# B&R Automation Studio project Haus
Automation Studio 4.8.4.50 SP; technology packages: mapp 5.13.1, mappView 5.13.1

## Configuration iCMSLight

CPU X20CP1586, AutomationRuntime B4.82, Build 4.1.2, Safety 0.0

### Task classes (Cpu.sw)
```
Cyclic#4 (cycle 32000 us, tolerance 32000 us):
  Solarpumpe <- Haus.Solarpumpe.prg
  Garage <- Haus.Garage.prg
  ErrorHandl <- Haus.ErrorHandling.prg
Cyclic#6 (cycle 256000 us, tolerance 256000 us):
  Main <- Haus.Main.prg
  Datenverwa <- Haus.Datenverwaltung.prg
DataObjects: assl3, Acp10sys, assl2, assl1
Binaries: TCLang, udbdef, mvLoader, TCData, arsvcreg, User, arconfig, Role, iomap, asfw, ashwac, ashwd, sysconf, Speicher, Units, RollenDB, Alarme, Config, VehicleAla, History, asnxdb2, OpcUaMap, MR4, Acp10map, acp10cfg, Shuttle2, MainAlarme, Alarm
Libraries: standard, runtime, operator, sys_lib, astime, brsystem, Convert, AsBrStr, ksTime, MpBase, FileIO, MpServer, AsMath, MpCom, MpRecipe, ksStpHist, DataObj, aruser, arssl, AsTCP, ksBuffer, AsOpcUac, AsHttp, MTBasics, AsHydCon, dvframe, MTTypes, AsUDP, ArCan, MTProfile, powerlnk, ksAlarm, MpAlarmX, AsSMTP, asstring
```

### Hardware
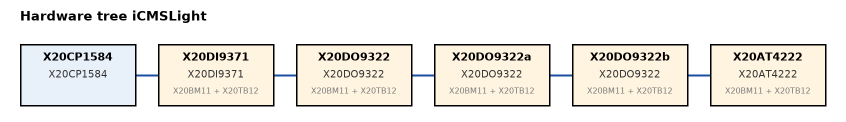
```
X20AT4222 : X20AT4222 v1.3.0.0  [SS1 -> X20TB12b.SS; SL -> X20BM11b.SL1]
  Supervision = off
  SensorType04 = off
X20BM11 : X20BM11 v1.0.0.1  [X2X1 -> X20BM11a.X2X2]
X20BM11a : X20BM11 v1.0.0.1  [X2X1 -> X20CP1584.IF6]
X20BM11b : X20BM11 v1.0.0.1  [X2X1 -> X20BM11d.X2X2]
X20BM11c : X20BM11 v1.0.0.1  [X2X1 -> X20BM11.X2X2]
X20BM11d : X20BM11 v1.0.0.1  [X2X1 -> X20BM11c.X2X2]
X20CP1584 : X20CP1584 v1.8.0.0
  Connector IF2:
    ActivateDevice = 1
    Mode = Manual
    InternetAddress = 192.168.0.101
    SubnetMask = 255.255.0.0
    ActivateOSAFT = 1
    OSAFTPortNumber = 10003
  Connector IF3:
    ActivatePowerlink = 0
  ConfigurationID = Haus
  SimulationModeOpcUa = off
  RemanentGlobalPvSize = 120652
  VolatileGlobalPvSize = 300000
  Connections = 10
  IdleTaskClass = 6
  TaskClassIdleTime = 10000
  CyclicTaskClassCount = 6
  Cyclic1Duration = 2000
  Cyclic1Tolerance = 2000
  Cyclic2Duration = 8000
  Cyclic2Tolerance = 8000
  Cyclic3Duration = 16000
  Cyclic3Tolerance = 16000
  Cyclic4Duration = 32000
  Cyclic4Tolerance = 32000
  Cyclic5Duration = 128000
  Cyclic5Tolerance = 128000
  Cyclic6Duration = 256000
  Cyclic6Tolerance = 256000
  FileDevice1
  FileDeviceName1 = Home
  FileDevicePath1 = C:\
  FileDevice2
  FileDeviceName2 = Alarm
  FileDevicePath2 = C:\Alarm
  FileDevice3
  FileDeviceName3 = Datenverwaltung
  FileDevicePath3 = C:\Datenverwaltung
  FileDevice4
  FileDeviceName4 = Logger
  FileDevicePath4 = C:\Logger
  TimeZone = 140
  ActivateDaylightSavingTime = 1
  FtpUser1
  FtpUsername1 = kssr
  FtpUserPassword1 = Z4sCxg1Qn6GbuX9/lK+IGbQPtWBLs+BxMSzu+/HSn5M=
  FtpUserSalt1 = QM4eEhG1
  FTPAccessRight1 = 0
  FTPdevice1 = ALL
  ActivateOpcUa = 1
  OpcUaLimitsMaxSessions = 0
  OpcUaLimitsMaxBrowseContinuationPoints = 50
  OpcUaInformationModels_PV_Version = 2
X20DI9371 : X20DI9371 v1.1.0.0  [SS1 -> X20TB12a.SS; SL -> X20BM11a.SL1]
  Supervision = off
X20DO9322 : X20DO9322 v1.2.0.0  [SS1 -> X20TB12.SS; SL -> X20BM11.SL1]
  Supervision = off
X20DO9322a : X20DO9322 v1.2.0.0  [SS1 -> X20TB12c.SS; SL -> X20BM11c.SL1]
  Supervision = off
X20DO9322b : X20DO9322 v1.2.0.0  [SS1 -> X20TB12d.SS; SL -> X20BM11d.SL1]
  Supervision = off
X20TB12 : X20TB12 v1.0.0.0
X20TB12a : X20TB12 v1.0.0.0
X20TB12b : X20TB12 v1.0.0.0
X20TB12c : X20TB12 v1.0.0.0
X20TB12d : X20TB12 v1.0.0.0
```

### IoMap.iom - X20CP1584/IoMap.iom
```iecst
VAR_CONFIG
	::Garage:IO.Output.Command AT %QX."X20DO9322".DigitalOutput01;
	::Garage:IO.Input.Opened AT %IX."X20DI9371".DigitalInput01;
	::Garage:IO.Input.Closed AT %IX."X20DI9371".DigitalInput02;
	::Solarpumpe:IO.Input.DachTemp AT %IW."X20AT4222".Temperature01;
	::Solarpumpe:IO.Input.RuecklaufTemp AT %IW."X20AT4222".Temperature02;
	::Solarpumpe:IO.Input.KesselTemp AT %IW."X20AT4222".Temperature03;
	::Garage:IO.Input.Button AT %IX."X20DI9371".DigitalInput03;
	::Solarpumpe:IO.Output.PumpeUp  AT %QX."X20DO9322a".DigitalOutput01;
	::Solarpumpe:IO.Output.PumpeDown  AT %QX."X20DO9322a".DigitalOutput02;
END_VAR
```

### Alarm.mpalarmxcore - X20CP1584/mappServices/Alarm.mpalarmxcore
```
Element gAlarmXCore (Type=mpalarmxcore)
  mapp.AlarmX.Core:
    Mapping:
      [0]
  mapp.AlarmX.Core.Configuration:
    [0]:
      Name = GarageUndefined
      Message = Das Garagentor ist in einem undefiniertem Zustand
      Behavior = PersistentAlarm
    [1]:
      Name = PumpUpNotActive
      Message = Die &#x2B06; Pumpe wurde nicht aktiviert da die Rücklauftemperatur zu hoch ist.
      Severity = 2
      Behavior = PersistentAlarm
  mapp.AlarmX.Core.Queries:
    [0]:
      Name = ActiveErrors
      Update = ::ErrorHandl:ActiveAlarms.Error.UpdateFlag
      Source:
        SELECT:
          [0]:
            Column = Severity
            PV = ::ErrorHandl:ActiveAlarms.Error.ActiveAlarms[]
        WHERE:
          [0]:
            Column = Severity
            CompareTo:
              Value = 1
    [1]:
      Name = ActiveWarnings
      Update = ::ErrorHandl:ActiveAlarms.Warning.UpdateFlag
      Source:
        SELECT:
          [0]:
            Column = Severity
            PV = ::ErrorHandl:ActiveAlarms.Warning.ActiveAlarms[]
        WHERE:
          [0]:
            Column = Severity
            CompareTo:
              Value = 2
    [2]:
      Name = ActiveInfos
      Update = ::ErrorHandl:ActiveAlarms.Info.UpdateFlag
      Source:
        SELECT:
          [0]:
            Column = Severity
            PV = ::ErrorHandl:ActiveAlarms.Info.ActiveAlarms[]
        WHERE:
          [0]:
            Column = Severity
            CompareTo:
              Value = 3
  mapp.AlarmX.Core.Categories:
    [0]:
      Name = Error
      SourceProperty:
        Severity = 1
    [1]:
      Name = Warning
      SourceProperty:
        Severity = 2
    [2]:
      Name = Info
      SourceProperty:
        Severity = 3
```

## Logical view

Binary libraries used (declarations not repeated): operator, runtime, astime, sys_lib, brsystem, standard, Convert, AsBrStr, ksTime 1.04.0, FileIO, AsMath, MpServer 5.13.0, MpBase 5.13.0, MpRecipe 5.13.1, MpCom 5.13.1, DataObj, MpAlarmX 5.11.2, AsSMTP, asstring

### Global.var - Global variables
```iecst
VAR
	gCurrentDT : DATE_AND_TIME := DT#1970-01-01-00:00:00;
	gSmtpSend : SmtpSend := (0);
	gCurrentDTStruct : DTStructure := (0);
END_VAR
```

### Package Logical/Libraries - Global libraries

### Library Logical/Libraries/ksStpHist (ANSIC, version 1.00.0) - Step History Baustein
Depends on: standard

#### ksStpHist.typ
```iecst
TYPE
	KsStepData_type : 	STRUCT
		Last : DINT;
		Act : DINT;
		Next : DINT; (*nur für single step*)
		Reset : DINT; (*step after reset*)
	END_STRUCT;
	ksStepHistoryEntry : 	STRUCT
		Act : USINT;
		ET : TIME;
	END_STRUCT;
END_TYPE
```

#### ksStpHist.fun
```iecst
{REDUND_ERROR} FUNCTION_BLOCK ksStepHistory (*speichert Schritthistorie*) (*$GROUP=User,$CAT=User,$GROUPICON=User.png,$CATICON=User.png*)
	VAR_INPUT
		in_Step : {REDUND_UNREPLICABLE} KsStepData_type;
		in_ET : {REDUND_UNREPLICABLE} TIME;
	END_VAR
	VAR
		aData : {REDUND_UNREPLICABLE} ARRAY[0..MAX_IDX_STEP_HISTORY_ENTRIES] OF ksStepHistoryEntry;
		i : {REDUND_UNREPLICABLE} USINT;
		Last : USINT;
	END_VAR
END_FUNCTION_BLOCK
```

#### ksStpHist.var
```iecst
VAR CONSTANT
	MAX_IDX_STEP_HISTORY_ENTRIES : USINT := 95;
END_VAR
```

#### ksStpHist.c
```c
#include <bur/plctypes.h>
#ifdef __cplusplus
	extern "C"
	{
#endif
	#include "ksStpHist.h"
#ifdef __cplusplus
	};
#endif
/* speichert Schritthistorie */
void ksStepHistory(struct ksStepHistory* inst)
{
	if (inst->i >= MAX_IDX_STEP_HISTORY_ENTRIES)
	{
		inst->i = 0;
	}

	if (inst->in_Step.Act != inst->in_Step.Next)
	{
		inst->aData[inst->i].Act = inst->in_Step.Act;
		inst->aData[inst->i].ET = inst->in_ET;
		inst->i++;
	}

}
```

### Program Logical/Haus/Main (ANSIC)

#### Main.c - Init, cyclic, exit code
```c
#include <bur/plctypes.h>
#include <stdbool.h>

#ifdef _DEFAULT_INCLUDES
	#include <AsDefault.h>
#endif

void _INIT ProgramInit(void)
{

}

void _CYCLIC ProgramCyclic(void)
{
	DTGetTime_1.enable = true;
	DTGetTime(&DTGetTime_1);

	gCurrentDT = DTGetTime_1.DT1;

	DT_TO_DTStructure(gCurrentDT, (UDINT)&gCurrentDTStruct);

	//Email Sender initialisieren

//	gSmtpSend.enable= true;
	gSmtpSend.pHost= (UDINT)"smtp.gmail.com";
	gSmtpSend.pSender= (UDINT)"sdillinger.tai@gmail.com";
	gSmtpSend.pReceiver= (UDINT)"mihawk14@web.de";
	gSmtpSend.pSubject= (UDINT)"test";
	gSmtpSend.pText= (UDINT)"test";
//	gSmtpSend.pUser = (UDINT)"sdillinger.tai@gmail.com";
//	gSmtpSend.pPassword= ADR(gMAIL.smpt_pw) // 'mein GMX Passwort'
//	gSmtpSend.pAttachment= ADR(AttStruc) // momentan 0
//	gSmtpSend.pDomain= 0
//	gSmtpSend.pSecurity= 0
//	gSmtpSend.timeout= 0
	gSmtpSend.port = 465; // 485,0, 0der 25
//	SmtpSend(&gSmtpSend);
}

void _EXIT ProgramExit(void)
{

}
```

#### Main.var - Local variables
```iecst
VAR
	DTGetTime_1 : DTGetTime := (0);
END_VAR
```

### Program Logical/Haus/Datenverwaltung (ANSIC)

#### Datenverwaltung.c - Init, cyclic, exit code
```c
#include <bur/plctypes.h>
#include <stdbool.h>
#include <AsBrStr.h>

#ifdef _DEFAULT_INCLUDES
	#include <AsDefault.h>
#endif

void _INIT ProgramInit(void)
{
    DirCreate_DV.enable = true;
    DirCreate_DV.pDevice = (UDINT)"Home";
    DirCreate_DV.pName = (UDINT)"Datenverwaltung";
    DirCreate(&DirCreate_DV);

    DTGetTime_DV.enable = true;
    DTGetTime(&DTGetTime_DV);

    Visu.StatusTime = DTGetTime_DV.DT1;
    brsstrcpy((UDINT)Visu.StatusText, (UDINT)"Steuerung neu gestartet");

    FileInfo_0.enable = true;
    FileInfo_0.pDevice = (UDINT)"Datenverwaltung";
    FileInfo_0.pName = (UDINT)"DV.csv";
    FileInfo_0.pInfo = (UDINT)&pFileInfo;
    FileInfo(&FileInfo_0);

    Visu.Load = true;

}

void _CYCLIC ProgramCyclic(void)
{
    DTGetTime_DV.enable = true;
    DTGetTime(&DTGetTime_DV);

    MpRecipeCsv_DV.MpLink = &gRecipeCsv;
    MpRecipeCsv_DV.Enable = true;
    MpRecipeCsv_DV.Save = Visu.Save;
    MpRecipeCsv_DV.Load = Visu.Load;
    MpRecipeCsv_DV.DeviceName = (UDINT)"Datenverwaltung";
    MpRecipeCsv_DV.FileName = (UDINT)"DV";
    MpRecipeCsv(&MpRecipeCsv_DV);

    for(i=0;i<=MAX_DV;i++)
    {
        MpRecipeRegPar_DV[i].MpLink = &gRecipeCsv;
        MpRecipeRegPar_DV[i].Enable = true;
        MpRecipeRegPar_DV[i].PVName = (UDINT)&PVNames[i];
        MpRecipeRegPar(&MpRecipeRegPar_DV[i]);
    }

    switch(State)
    {
        case STATE_DV_WAIT:
            Visu.ButtonAktiv = true;
            if(Visu.Save)
            {
                Visu.ButtonAktiv = false;
                State = STATE_DV_SAVE;
            }
            else if(Visu.Load)
            {
                Visu.ButtonAktiv = false;
                State = STATE_DV_LOAD;
            }

            break;

        case STATE_DV_SAVE:
            if(MpRecipeCsv_DV.CommandDone)
            {
                Visu.StatusTime = DTGetTime_DV.DT1;
                brsstrcpy((UDINT)Visu.StatusText, (UDINT)"Speichern abgeschlossen");
                Visu.Save = false;
                State = STATE_DV_WAIT;
            }

            break;

        case STATE_DV_LOAD:
            if(MpRecipeCsv_DV.CommandDone)
            {
                Visu.StatusTime = DTGetTime_DV.DT1;
                brsstrcpy((UDINT)Visu.StatusText, (UDINT)"Laden abgeschlossen");
                Visu.Load = false;
                State = STATE_DV_WAIT;
            }

            break;

    }

}

void _EXIT ProgramExit(void)
{
    MpRecipeCsv_DV.Enable = false;
    MpRecipeCsv(&MpRecipeCsv_DV);

//    for(i=0;i<=MAX_DV;i++)
//    {
//        MpRecipeRegPar_DV[i].Enable = false;
//        MpRecipeRegPar(&MpRecipeRegPar_DV[i]);
//    }
}
```

#### Datenverwaltung.typ - Local data types
```iecst
TYPE
	STATE_DV_enum :
		(
		STATE_DV_WAIT,
		STATE_DV_SAVE,
		STATE_DV_LOAD
		);
	DatenverwaltungVisu_typ : 	STRUCT
		Save : BOOL;
		Load : BOOL;
		ButtonAktiv : BOOL;
		StatusText : STRING[255];
		StatusTime : DATE_AND_TIME;
	END_STRUCT;
END_TYPE
```

#### Datenverwaltung.var - Local variables
```iecst
VAR CONSTANT
	MAX_DV : USINT := 10;
END_VAR
VAR
	MpRecipeRegPar_DV : ARRAY[0..MAX_DV] OF MpRecipeRegPar := [11((0))];
	MpRecipeCsv_DV : MpRecipeCsv := (0);
	PVNames : ARRAY[0..MAX_DV] OF STRING[255] := ['Solarpumpe:DachSollTemp','Solarpumpe:KesselSollTemp','Solarpumpe:RuecklaufSollTemp','RuecklaufTimeOffset',7('')];
	DTGetTime_DV : DTGetTime := (0);
	DirCreate_DV : DirCreate := (0);
	i : USINT := 0;
	Visu : DatenverwaltungVisu_typ := (0);
	State : STATE_DV_enum := STATE_DV_WAIT;
	FileInfo_0 : FileInfo := (0);
	pFileInfo : REFERENCE TO fiFILE_INFO;
END_VAR
```

### Program Logical/Haus/Solarpumpe (ANSIC)

#### Solarpumpe.c - Init, cyclic, exit code
```c
#include <bur/plctypes.h>
#include <stdbool.h>

#ifdef _DEFAULT_INCLUDES
	#include <AsDefault.h>
#endif

void _INIT ProgramInit(void)
{

}

void _CYCLIC ProgramCyclic(void)
{
	if(IO.Output.PumpeDown)
		brsstrcpy((UDINT)Visu.PumpeDownStyle, (UDINT)"StatusOk");
	else
		brsstrcpy((UDINT)Visu.PumpeDownStyle, (UDINT)"StatusNOk");

	if(IO.Output.PumpeUp)
		brsstrcpy((UDINT)Visu.PumpeUpStyle, (UDINT)"StatusOk");
	else
		brsstrcpy((UDINT)Visu.PumpeUpStyle, (UDINT)"StatusNOk");

	UDINTTimeOffset = Mem.RuecklaufTimeOffset;

	TON_PumpUp.IN = IO.Output.PumpeDown;
	TON_PumpUp.PT = UDINTTimeOffset * 1000;
	TON(&TON_PumpUp);

	R_TRIG_Start.CLK = IO.Output.PumpeUp && IO.Output.PumpeDown;
	R_TRIG(&R_TRIG_Start);

	R_TRIG_Stop.CLK = !(IO.Output.PumpeUp && IO.Output.PumpeDown);
	R_TRIG(&R_TRIG_Stop);

	if(R_TRIG_Start.Q)
	{
		Info.LastStart = gCurrentDT;
	}

	if(R_TRIG_Stop.Q)
	{
	 	Info.LastStop = gCurrentDT;
		Info.LaufzeitDownAkt = 0;
		Info.LaufzeitUpAkt = 0;
	}

	if(Mem.Aktiv)
	{
		if(IO.Input.DachTemp >= Mem.DachSollTemp && IO.Input.KesselTemp <= Mem.KesselSollTemp)
		{
			IO.Output.PumpeDown = true;
			Info.LaufzeitDownAkt += CURRENT_CYCLE_TIME;
			Info.LaufzeitUpGes += CURRENT_CYCLE_TIME;

			if(TON_PumpUp.Q)
			{
				if(IO.Input.RuecklaufTemp <= Mem.RuecklaufSollTemp)
				{
					IO.Output.PumpeUp = true;
					Info.LaufzeitUpAkt += CURRENT_CYCLE_TIME;
					Info.LaufzeitDownGes += CURRENT_CYCLE_TIME;

					MpAlarmXReset(&gAlarmXCore, "PumpUpNotActive");
				}
				else
				{
					MpAlarmXSet(&gAlarmXCore, "PumpUpNotActive");
				}
			}
		}
		else
		{
			IO.Output.PumpeDown = false;
			IO.Output.PumpeUp = false;
		}

	}
	else
	{
		IO.Output.PumpeDown = false;
		IO.Output.PumpeUp = false;
	}
}

void _EXIT ProgramExit(void)
{

}
```

#### Solarpumpe.typ - Local data types
```iecst
TYPE
	SolarpumpeIO_typ : 	STRUCT
		Input : SolarpumpeInputs_typ;
		Output : SolarpumpeOutputs_typ;
	END_STRUCT;
	SolarpumpeInputs_typ : 	STRUCT
		DachTemp : INT;
		RuecklaufTemp : INT;
		KesselTemp : INT;
	END_STRUCT;
	SolarpumpeOutputs_typ : 	STRUCT
		PumpeDown : BOOL;
		PumpeUp : BOOL;
	END_STRUCT;
	SolarpumpeVisu_typ : 	STRUCT
		PumpeUpStyle : STRING[99];
		PumpeDownStyle : STRING[99];
	END_STRUCT;
	SolarpumpeInfo_typ : 	STRUCT
		LaufzeitDownAkt : DINT;
		LaufzeitUpAkt : DINT;
		LaufzeitDownGes : DINT;
		LaufzeitUpGes : DINT;
		LastStart : DATE_AND_TIME;
		LastStop : DATE_AND_TIME;
	END_STRUCT;
	SolarpumpeMem_typ : 	STRUCT
		DachSollTemp : INT;
		KesselSollTemp : INT;
		RuecklaufSollTemp : INT;
		Aktiv : BOOL;
		RuecklaufTimeOffset : DATE_AND_TIME;
	END_STRUCT;
END_TYPE
```

#### Solarpumpe.var - Local variables
```iecst
VAR
	IO : SolarpumpeIO_typ := (0);
	Mem : SolarpumpeMem_typ := (0);
	Visu : SolarpumpeVisu_typ := (0);
	TON_PumpUp : TON := (0);
	UDINTTimeOffset : UDINT := 0;
	Info : SolarpumpeInfo_typ := (0);
	R_TRIG_Start : R_TRIG := (0);
	R_TRIG_Stop : R_TRIG := (0);
END_VAR
VAR CONSTANT
	CURRENT_CYCLE_TIME : USINT := 32;
END_VAR
```

### Program Logical/Haus/Garage (ANSIC)

#### Garage.c - Init, cyclic, exit code
```c
#include <bur/plctypes.h>
#include <stdbool.h>

#ifdef _DEFAULT_INCLUDES
	#include <AsDefault.h>
#endif

void _INIT ProgramInit(void)
{

}

void _CYCLIC ProgramCyclic(void)
{

	DT_TO_DTStructure(Mem.Schliesszeit, (UDINT)&Mem.SchliesszeitStruct);

	IO.Output.Command = IO.Input.Button || Stat.AutoClose;

	if(IO.Input.Closed || IO.Input.Opened)
	{
		Visu.ButtonActiveOpen = IO.Input.Closed;
		Visu.ButtonActiveClose = IO.Input.Opened;
	}
	else
	{
		Visu.ButtonActiveOpen = true;
		Visu.ButtonActiveClose = true;
	}

	if(Mem.Automatik)
	{
		if(Mem.Nachlaufzeit != 0)
		{
			Stat.TON_Nachlaufzeit.IN = IO.Input.Opened;
			Stat.TON_Nachlaufzeit.PT = Mem.Nachlaufzeit;
			TON(&Stat.TON_Nachlaufzeit);
		}
		else
		{
			Stat.TON_Nachlaufzeit.IN = false;
			TON(&Stat.TON_Nachlaufzeit);
		}

		if((Mem.SchliesszeitStruct.hour == gCurrentDTStruct.hour &&
			Mem.SchliesszeitStruct.minute == gCurrentDTStruct.minute &&
			Mem.SchliesszeitStruct.second == gCurrentDTStruct.second) ||
			Stat.TON_Nachlaufzeit.Q)
		{
			Stat.AutoClose = true;
		}
		else
		{
			Stat.AutoClose = false;
		}

	}
	else
	{
		Stat.AutoClose = false;
	}

}

void _EXIT ProgramExit(void)
{

}
```

#### Garage.typ - Local data types
```iecst
TYPE
	GarageIO_typ : 	STRUCT
		Input : GarageInput_typ;
		Output : GarageOutput_typ;
	END_STRUCT;
	GarageStat_typ : 	STRUCT
		AutoClose : BOOL;
		TON_Nachlaufzeit : TON;
	END_STRUCT;
	GarageMem_typ : 	STRUCT
		Schliesszeit : DATE_AND_TIME;
		SchliesszeitStruct : DTStructure;
		Nachlaufzeit : DINT;
		Automatik : BOOL;
	END_STRUCT;
	GarageInput_typ : 	STRUCT
		Opened : BOOL;
		Closed : BOOL;
		Button : BOOL;
	END_STRUCT;
	GarageOutput_typ : 	STRUCT
		Command : BOOL;
	END_STRUCT;
	GarageVisu_typ : 	STRUCT
		ButtonActiveOpen : BOOL;
		ButtonActiveClose : BOOL;
	END_STRUCT;
END_TYPE
```

#### Garage.var - Local variables
```iecst
VAR
	Mem : GarageMem_typ := (0);
	IO : GarageIO_typ := (0);
	Stat : GarageStat_typ := (0);
	Visu : GarageVisu_typ := (0);
END_VAR
```

### Program Logical/Haus/ErrorHandling (ANSIC)

#### ErrorHandling.c - Init, cyclic, exit code
```c
#include <bur/plctypes.h>
#include <stdbool.h>
#include <string.h>
#include <AsBrStr.h>

#ifdef _DEFAULT_INCLUDES
#include <AsDefault.h>
#endif

void _INIT ProgramInit(void)
{
//	MpAlarmXSet(&gAlarmXCore, StackerAlarmStrings[z].Name[i]);
//
//	MpAlarmXReset(&gAlarmXCore, StackerAlarmStrings[z].Name[i]);

}

void _CYCLIC ProgramCyclic(void)
{
    /* Alarmsystem */
    MpAlarmXCore_1.MpLink = &gAlarmXCore;
    MpAlarmXCore_1.Enable = true;
    MpAlarmXCore_1.ErrorReset = ResetMpError;
    MpAlarmXCore(&MpAlarmXCore_1);

    Visu.AlarmVisible = (MpAlarmXCore_1.PendingAlarms != 0);

    // AlarmConfig
    brsstrcpy((UDINT)Visu.AlarmConfigString, (UDINT)ALARMLIST_CONFIG);

    // Überprüfen welche Severities aktiv sind
    Visu.ErrorAktiv = false;
    Visu.WarningAktiv = false;
    Visu.InfoAktiv = false;
    if(MpAlarmXCheckReaction(&gAlarmXCore, "ErrorAktiv"))
        Visu.ErrorAktiv = true;
    else if(MpAlarmXCheckReaction(&gAlarmXCore, "WarningAktiv"))
        Visu.WarningAktiv = true;
    else if(MpAlarmXCheckReaction(&gAlarmXCore, "InfoAktiv"))
        Visu.InfoAktiv = true;

    // Auswertung Aktiver Alarme
    // Error
    MpAlarmXQuery_0.MpLink = &gAlarmXCore;;
    MpAlarmXQuery_0.Enable = true;
    MpAlarmXQuery_0.ErrorReset = ResetMpError;
    MpAlarmXQuery_0.Mode = mpALARMX_QUERY_MODE_ALL ;
    MpAlarmXQuery_0.Name = (UDINT)"ActiveErrors";
    MpAlarmXQuery_0.Execute = (ActiveAlarms.Error.UpdateFlag != ActiveAlarms.Error.UpdateFlagOld);
    MpAlarmXQuery(&MpAlarmXQuery_0);

    if(MpAlarmXQuery_0.CommandDone)
    {
        ActiveAlarms.Error.Count = MpAlarmXQuery_0.Info.RowsRead;
        ActiveAlarms.Error.UpdateFlagOld = ActiveAlarms.Error.UpdateFlag;
    }

    // Warning
    MpAlarmXQuery_1.MpLink = &gAlarmXCore;;
    MpAlarmXQuery_1.Enable = true;
    MpAlarmXQuery_1.ErrorReset = ResetMpError;
    MpAlarmXQuery_1.Mode = mpALARMX_QUERY_MODE_ALL ;
    MpAlarmXQuery_1.Name = (UDINT)"ActiveWarnings";
    MpAlarmXQuery_1.Execute = (ActiveAlarms.Warning.UpdateFlag != ActiveAlarms.Warning.UpdateFlagOld);
    MpAlarmXQuery(&MpAlarmXQuery_1);

    if(MpAlarmXQuery_1.CommandDone)
    {
        ActiveAlarms.Warning.Count = MpAlarmXQuery_1.Info.RowsRead;
        ActiveAlarms.Warning.UpdateFlagOld = ActiveAlarms.Warning.UpdateFlag;
    }

    // Info
    MpAlarmXQuery_2.MpLink = &gAlarmXCore;;
    MpAlarmXQuery_2.Enable = true;
    MpAlarmXQuery_2.ErrorReset = ResetMpError;
    MpAlarmXQuery_2.Mode = mpALARMX_QUERY_MODE_ALL ;
    MpAlarmXQuery_2.Name = (UDINT)"ActiveInfos";
    MpAlarmXQuery_2.Execute = (ActiveAlarms.Info.UpdateFlag != ActiveAlarms.Info.UpdateFlagOld);
    MpAlarmXQuery(&MpAlarmXQuery_2);

    if(MpAlarmXQuery_2.CommandDone)
    {
        ActiveAlarms.Info.Count = MpAlarmXQuery_2.Info.RowsRead;
        ActiveAlarms.Info.UpdateFlagOld = ActiveAlarms.Info.UpdateFlag;
    }

    ActiveAlarms.CountAll = ActiveAlarms.Error.Count + ActiveAlarms.Warning.Count + ActiveAlarms.Info.Count;
    ActiveAlarms.Visible = (ActiveAlarms.CountAll != 0);

    if(Visu.ErrorAktiv)
        brsstrcpy((UDINT)Visu.FooterImage, (UDINT)"Media/Images/BHS/Alarme/224_Warning_act.svg");
    else if(Visu.WarningAktiv)
        brsstrcpy((UDINT)Visu.FooterImage, (UDINT)"Media/Images/BHS/Alarme/226_Attention_act.svg");
    else if(Visu.InfoAktiv)
        brsstrcpy((UDINT)Visu.FooterImage, (UDINT)"Media/Images/BHS/Alarme/180_Maintenance_act.svg");
    else
        brsstrcpy((UDINT)Visu.FooterImage, (UDINT)"Media/Images/BHS/Alarme/224_Warning_ena.svg");

}

void _EXIT ProgramExit(void)
{
    MpAlarmXCore_1.Enable = false;
    MpAlarmXCore(&MpAlarmXCore_1);
}
```

#### ErrorHandling.typ - Local data types
```iecst
TYPE
	ErrorHandlingVisu_typ : 	STRUCT
		AlarmVisible : BOOL;
		ErrorAktiv : BOOL;
		WarningAktiv : BOOL;
		InfoAktiv : BOOL;
		AlarmConfigString : STRING[1000];
		FooterImage : STRING[255];
	END_STRUCT;
	ActiveAlarms_type : 	STRUCT
		Error : ActiveAlarmsConfig_type;
		Warning : ActiveAlarmsConfig_type;
		Info : ActiveAlarmsConfig_type;
		CountAll : UINT;
		Visible : BOOL;
	END_STRUCT;
	ActiveAlarmsConfig_type : 	STRUCT
		UpdateFlag : UDINT;
		UpdateFlagOld : UDINT;
		ActiveAlarms : ARRAY[0..999]OF STRING[100];
		Count : UINT;
	END_STRUCT;
END_TYPE
```

#### ErrorHandling.var - Local variables
```iecst
VAR CONSTANT
	ALARMLIST_CONFIG : STRING[1000] := '[{"styleNbr":1,"alarmState":5,"severity":[{"useState":true,"value":1,"conditionType":"=="},{"useState":false,"value":0,"conditionType":">"}]},{"styleNbr":2,"alarmState":5,"severity":[{"useState":true,"value":2,"conditionType":"=="},{"useState":false,"value":0,"conditionType":">"}]},{"styleNbr":3,"alarmState":5,"severity":[{"useState":true,"value":3,"conditionType":"=="},{"useState":false,"value":0,"conditionType":">"}]}]';
END_VAR
VAR
	MpAlarmXCore_1 : MpAlarmXCore;
	ResetMpError : BOOL;
	Visu : ErrorHandlingVisu_typ := (0);
	MpAlarmXQuery_1 : MpAlarmXQuery := (0);
	MpAlarmXQuery_2 : MpAlarmXQuery := (0);
	MpAlarmXQuery_0 : MpAlarmXQuery := (0);
	ActiveAlarms : ActiveAlarms_type := (0);
END_VAR
```

- Project.language (not shown)

- Visualisation Logical/mappView (not shown)

Listed in the project but not available here: Logical/Global.typ, Logical/GlobalConst.var, Logical/Haus/Main/Main.typ
